(*
Rounds the input signal to the nearest multiple of :attr:`StepSize`.

Useful for simulating ADC resolution, modelling actuators with discrete
positions, or testing controller behaviour under quantisation.

A :attr:`StepSize` of zero passes the input through unchanged.

.. note::
   The block is ``FINAL`` and must be instantiated, not extended.
   Use ``FB_init`` to set :attr:`fStepSize` at declaration time.
*)
{attribute 'enable_dynamic_creation'}
{attribute 'no_explicit_call' := 'direct call for this function block is not allowed'}
FUNCTION_BLOCK FINAL FB_Quantizer EXTENDS FB_SisoComponent
IMPLEMENTS FsCommon.I_Runnable
VAR
	_fStepSize : LREAL; // Quantisation step size. Zero passes the input through unchanged.
END_VAR

METHOD FB_init : BOOL
VAR_INPUT
	bInitRetains : BOOL; // if TRUE, the retain variables are initialized (warm start / cold start)
	bInCopyCode  : BOOL;  // if TRUE, the instance afterwards gets moved into the copy code (online change)
	fStepSize    : LREAL; // Quantisation step size. Zero passes the input through unchanged.
END_VAR
THIS^._fStepSize := fStepSize;
END_METHOD

(* Applies quantisation to the current input. *)
METHOD Run
VAR_INPUT
END_VAR
IF THIS^._fStepSize = 0 THEN
	THIS^._fOutput := THIS^._fInput;
	RETURN;
END_IF

THIS^._fOutput := FsCommon.F_TruncateNumber(
	THIS^._fInput / THIS^._fStepSize + 0.5
) * THIS^._fStepSize;
END_METHOD

(*
Gets or sets the quantisation step size.

The output is rounded to the nearest multiple of this value. For example,
a step size of 0.5 rounds the input to the nearest 0.5. A value of zero
passes the input through unchanged.
*)
PROPERTY StepSize : LREAL
GET
StepSize := THIS^._fStepSize;
END_GET
SET
THIS^._fStepSize := StepSize;
END_SET
END_PROPERTY

END_FUNCTION_BLOCK

(* stored: Version 1.1.0.1, ProductVersion 3.1.4024.15
   POU FB_Quantizer: Id {f6873a72-5b17-40ab-a215-a99a0df1449b}, SpecialFunc None
   Method FB_init: Id {fa282ad0-d329-46b7-8d76-c4303520d801}
   Method Run: Id {849f905a-d254-4e5d-bc42-9c82dac4dfc1}
   Property StepSize: Id {40436987-be23-4e42-a609-af08620aeba2}
   Get Get: Id {7230e5e7-827a-4094-9b15-bae9c2480703}
   Set Set: Id {8fd83605-6030-4988-aa87-1e7d956ff7e2} *)
